(* PLC project  *)

PROGRAM P

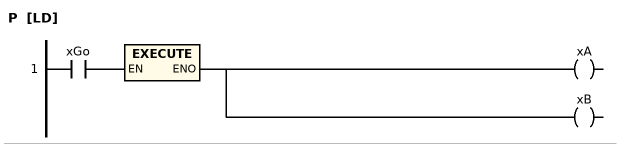
(* LD diagram, written out as Structured Text *)
IF xGo THEN
  nCount := nCount + 1;
END_IF;
xA := xGo;
xB := xGo;
END_PROGRAM
